(* Schneider Machine Expert - Basic project Prototype 3, file version 2.7.0.0 *)
(* ProjectInformations: Name=Nuevo proyecto *)

HARDWARE
  Cpu 0: TM221M16R/G
  EthernetConfiguration: NetworkName=M221, IpAllocationMode=FixedAddress, IpAddress=0.0.0.0, SubnetMask=0.0.0.0
  SerialLineConfiguration: Baud=Baud19200, Parity=ParityEven, DataBits=DataBits8, StopBits=StopBits1, PhysicalMedium=PhysicalMediumRs485, TransmissionMode=TransmissionModeModbusRtu, SlaveId=1, Addressing=SlaveAddressing
  MastTask: UsePeriodScanMode=false, PeriodScan=100
  FastTask: Period=255
  CpuBehavior: StartingMode=StartAsPreviousState, AutoSaveRamOnEeprom=true, WatchdogPeriod=250

SYMBOLS  (address, symbol, comment, settings)
  %M0       START_BUTTON
  %M1       FINISH_BUTTON
  %M2       STOP_BUTTON
  %M3       EMERGENCY_STOP
  %M4       TYPE_2
  %M5       TYPE_3
  %M6       MACHINE_2
  %M7       MACHINE_3
  %M8       ITEM_1
  %M9       DOOR
  %M10      EXIT_PROCESS_SENSOR
  %M11      ITEM_2
  %M12      RESET_BUTTON
  %M13      ALARM_SIREN
  %M14      GREEN_LIGHT
  %M15      YELLOW_LIGHT
  %M16      RED_LIGHT
  %M17      WARNING_LIGHT
  %M18      GRAB_1
  %M19      PROCESS_INIT
  %M20      AUX_CONVEYOR
  %M21      PROCESS_EXIT
  %M22      GRAB_2
  %M100     INIT_1
  %M200     OK
  %S21      SB_INITGRAFCET  "En el estado 1, este bit provoca una inicialización GRAFCET. Los pasos activos se desactivan y los pasos iniciales se activan"
  %X1       STATE_1
  %X2       STATE_2
  %X3       STATE_3
  %X4       STATE_4
  %X5       STATE_5
  %X6       STATE_6
  %X7       STATE_7
  %X8       STATE_8
  %X9       STATE_9
  %X11      STATE_11
  %X12      STATE_12
  %X13      STATE_13
  %X14      STATE_14
  %X15      STATE_15
  %X17      STATE_17
  %X18      STATE_18
  %X19      STATE_19
  %X20      STATE_20
  %MW0      X_1
  %MW1      Y_1
  %MW2      Z_1
  %MW3      X_2
  %MW4      Y_2
  %MW5      Z_2
  %MW6      SET_X_1
  %MW7      SET_Y_1
  %MW8      SET_Z_1
  %MW9      SET_X_2
  %MW10     SET_Y_2
  %MW11     SET_Z_2
  %MW12     M1
  %MW13     M2
  %MW14     M3
  %KF1      X_Y_ZERO  [Value=0]
  %KF4      X_Y_MED  [Value=5.1]
  %KF7      X_Y_MAX  [Value=10]
  %KF10     Z_MAX  [Value=5.9]
  %KF13     Z_MIN  [Value=2.5]
  %KF16     TOL  [Value=0.1]
  %TM0      SECURITY_TIME  [Preset=5, Base=OneSecond]
  %TM1      FINISH_CONEYOR  [Type=TOF, Preset=3, Base=OneSecond]
  %C0       MACHINE_1_INPUT  [Preset=1000]
  %C1       MACHINE_2_INPUT  [Preset=1000]
  %C2       MACHINE_3_INPUT  [Preset=1000]

GRAFCET Grafcet
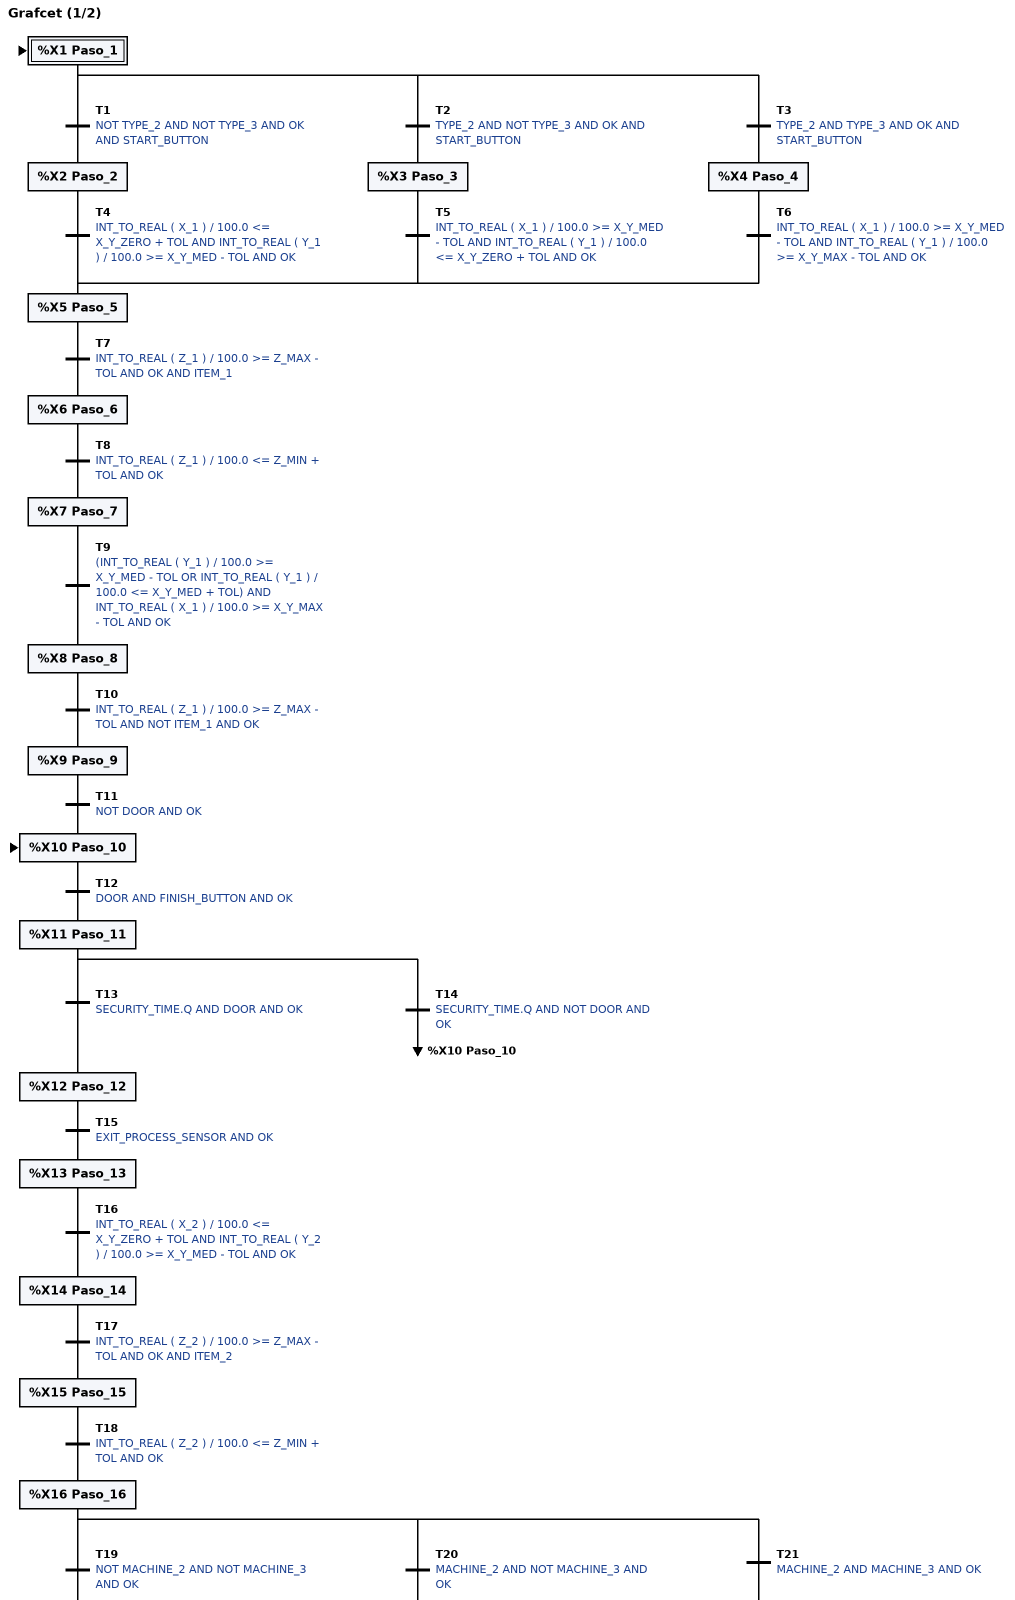
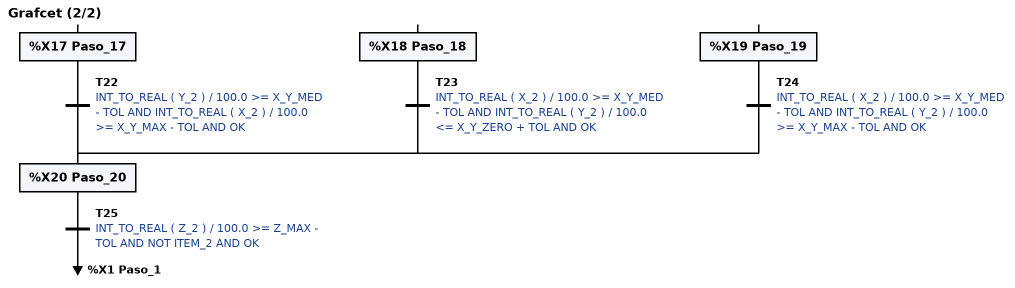
  INITIAL_STEP %X1  (* Paso_1 *)
  STEP %X2  (* Paso_2 *)
  STEP %X3  (* Paso_3 *)
  STEP %X4  (* Paso_4 *)
  STEP %X5  (* Paso_5 *)
  STEP %X6  (* Paso_6 *)
  STEP %X7  (* Paso_7 *)
  STEP %X8  (* Paso_8 *)
  STEP %X9  (* Paso_9 *)
  STEP %X10  (* Paso_10 *)
  STEP %X11  (* Paso_11 *)
  STEP %X12  (* Paso_12 *)
  STEP %X13  (* Paso_13 *)
  STEP %X14  (* Paso_14 *)
  STEP %X15  (* Paso_15 *)
  STEP %X16  (* Paso_16 *)
  STEP %X17  (* Paso_17 *)
  STEP %X18  (* Paso_18 *)
  STEP %X19  (* Paso_19 *)
  STEP %X20  (* Paso_20 *)
  TRANSITION T1 FROM %X1 TO %X2 := NOT TYPE_2 AND NOT TYPE_3 AND OK AND START_BUTTON;
  TRANSITION T2 FROM %X1 TO %X3 := TYPE_2 AND NOT TYPE_3 AND OK AND START_BUTTON;
  TRANSITION T3 FROM %X1 TO %X4 := TYPE_2 AND TYPE_3 AND OK AND START_BUTTON;
  TRANSITION T4 FROM %X2 TO %X5 := INT_TO_REAL ( X_1 ) / 100.0 <= X_Y_ZERO + TOL AND INT_TO_REAL ( Y_1 ) / 100.0 >= X_Y_MED - TOL AND OK;
  TRANSITION T5 FROM %X3 TO %X5 := INT_TO_REAL ( X_1 ) / 100.0 >= X_Y_MED - TOL AND INT_TO_REAL ( Y_1 ) / 100.0 <= X_Y_ZERO + TOL AND OK;
  TRANSITION T6 FROM %X4 TO %X5 := INT_TO_REAL ( X_1 ) / 100.0 >= X_Y_MED - TOL AND INT_TO_REAL ( Y_1 ) / 100.0 >= X_Y_MAX - TOL AND OK;
  TRANSITION T7 FROM %X5 TO %X6 := INT_TO_REAL ( Z_1 ) / 100.0 >= Z_MAX - TOL AND OK AND ITEM_1;
  TRANSITION T8 FROM %X6 TO %X7 := INT_TO_REAL ( Z_1 ) / 100.0 <= Z_MIN + TOL AND OK;
  TRANSITION T9 FROM %X7 TO %X8 := (INT_TO_REAL ( Y_1 ) / 100.0 >= X_Y_MED - TOL OR INT_TO_REAL ( Y_1 ) / 100.0 <= X_Y_MED + TOL) AND INT_TO_REAL ( X_1 ) / 100.0 >= X_Y_MAX - TOL AND OK;
  TRANSITION T10 FROM %X8 TO %X9 := INT_TO_REAL ( Z_1 ) / 100.0 >= Z_MAX - TOL AND NOT ITEM_1 AND OK;
  TRANSITION T11 FROM %X9 TO %X10 := NOT DOOR AND OK;
  TRANSITION T12 FROM %X10 TO %X11 := DOOR AND FINISH_BUTTON AND OK;
  TRANSITION T13 FROM %X11 TO %X12 := SECURITY_TIME.Q AND DOOR AND OK;
  TRANSITION T14 FROM %X11 TO %X10 := SECURITY_TIME.Q AND NOT DOOR AND OK;
  TRANSITION T15 FROM %X12 TO %X13 := EXIT_PROCESS_SENSOR AND OK;
  TRANSITION T16 FROM %X13 TO %X14 := INT_TO_REAL ( X_2 ) / 100.0 <= X_Y_ZERO + TOL AND INT_TO_REAL ( Y_2 ) / 100.0 >= X_Y_MED - TOL AND OK;
  TRANSITION T17 FROM %X14 TO %X15 := INT_TO_REAL ( Z_2 ) / 100.0 >= Z_MAX - TOL AND OK AND ITEM_2;
  TRANSITION T18 FROM %X15 TO %X16 := INT_TO_REAL ( Z_2 ) / 100.0 <= Z_MIN + TOL AND OK;
  TRANSITION T19 FROM %X16 TO %X17 := NOT MACHINE_2 AND NOT MACHINE_3 AND OK;
  TRANSITION T20 FROM %X16 TO %X18 := MACHINE_2 AND NOT MACHINE_3 AND OK;
  TRANSITION T21 FROM %X16 TO %X19 := MACHINE_2 AND MACHINE_3 AND OK;
  TRANSITION T22 FROM %X17 TO %X20 := INT_TO_REAL ( Y_2 ) / 100.0 >= X_Y_MED - TOL AND INT_TO_REAL ( X_2 ) / 100.0 >= X_Y_MAX - TOL AND OK;
  TRANSITION T23 FROM %X18 TO %X20 := INT_TO_REAL ( X_2 ) / 100.0 >= X_Y_MED - TOL AND INT_TO_REAL ( Y_2 ) / 100.0 <= X_Y_ZERO + TOL AND OK;
  TRANSITION T24 FROM %X19 TO %X20 := INT_TO_REAL ( X_2 ) / 100.0 >= X_Y_MED - TOL AND INT_TO_REAL ( Y_2 ) / 100.0 >= X_Y_MAX - TOL AND OK;
  TRANSITION T25 FROM %X20 TO %X1 := INT_TO_REAL ( Z_2 ) / 100.0 >= Z_MAX - TOL AND NOT ITEM_2 AND OK;

TRANSITION T1 (%X1 -> %X2) 
  (* SectionNumber=0 *)

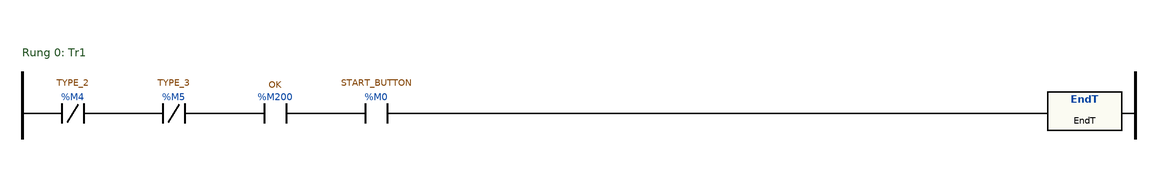

// Rung 0: Tr1
  LDN %M4                 (* TYPE_2 *)
  ANDN %M5                (* TYPE_3 *)
  AND %M200               (* OK *)
  AND %M0                 (* START_BUTTON *)
  ENDT
  // as ST:
  //   TRANSITION := NOT TYPE_2 AND NOT TYPE_3 AND OK AND START_BUTTON;

TRANSITION T2 (%X1 -> %X3) 
  (* SectionNumber=0 *)

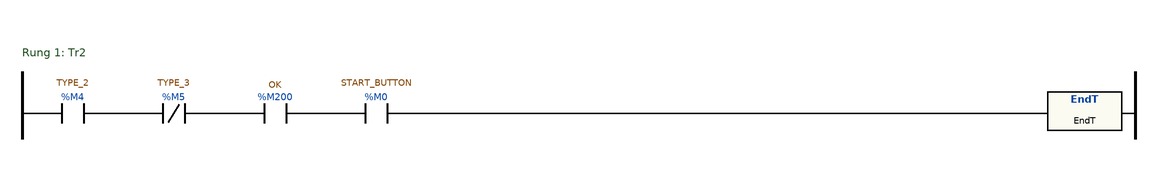

// Rung 1: Tr2
  LD %M4                  (* TYPE_2 *)
  ANDN %M5                (* TYPE_3 *)
  AND %M200               (* OK *)
  AND %M0                 (* START_BUTTON *)
  ENDT
  // as ST:
  //   TRANSITION := TYPE_2 AND NOT TYPE_3 AND OK AND START_BUTTON;

TRANSITION T3 (%X1 -> %X4) 
  (* SectionNumber=0 *)

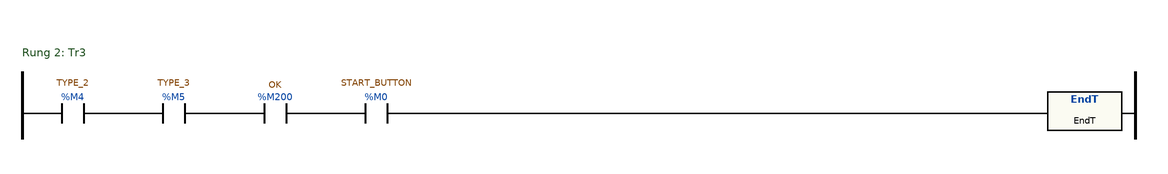

// Rung 2: Tr3
  LD %M4                  (* TYPE_2 *)
  AND %M5                 (* TYPE_3 *)
  AND %M200               (* OK *)
  AND %M0                 (* START_BUTTON *)
  ENDT
  // as ST:
  //   TRANSITION := TYPE_2 AND TYPE_3 AND OK AND START_BUTTON;

TRANSITION T4 (%X2 -> %X5) 
  (* SectionNumber=0 *)

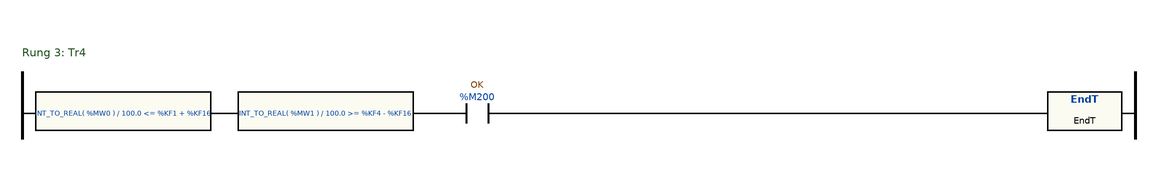

// Rung 3: Tr4
  LD 1
  AND [ INT_TO_REAL ( %MW0 ) / 100.0 <= %KF1 + %KF16 ](* X_1, X_Y_ZERO, TOL *)
  AND [ INT_TO_REAL ( %MW1 ) / 100.0 >= %KF4 - %KF16 ](* Y_1, X_Y_MED, TOL *)
  AND %M200               (* OK *)
  ENDT
  // as ST:
  //   TRANSITION := INT_TO_REAL ( X_1 ) / 100.0 <= X_Y_ZERO + TOL AND INT_TO_REAL ( Y_1 ) / 100.0 >= X_Y_MED - TOL AND OK;

TRANSITION T5 (%X3 -> %X5) 
  (* SectionNumber=0 *)

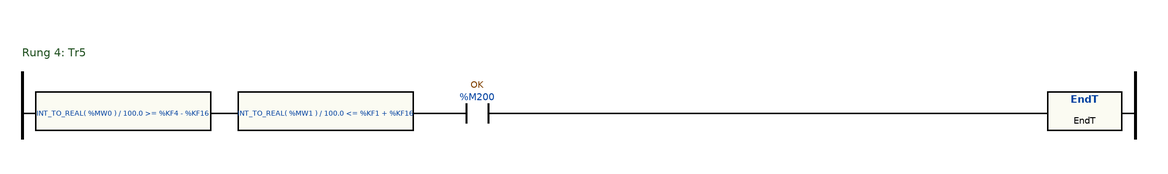

// Rung 4: Tr5
  LD 1
  AND [ INT_TO_REAL ( %MW0 ) / 100.0 >= %KF4 - %KF16 ](* X_1, X_Y_MED, TOL *)
  AND [ INT_TO_REAL ( %MW1 ) / 100.0 <= %KF1 + %KF16 ](* Y_1, X_Y_ZERO, TOL *)
  AND %M200               (* OK *)
  ENDT
  // as ST:
  //   TRANSITION := INT_TO_REAL ( X_1 ) / 100.0 >= X_Y_MED - TOL AND INT_TO_REAL ( Y_1 ) / 100.0 <= X_Y_ZERO + TOL AND OK;

TRANSITION T6 (%X4 -> %X5) 
  (* SectionNumber=0 *)

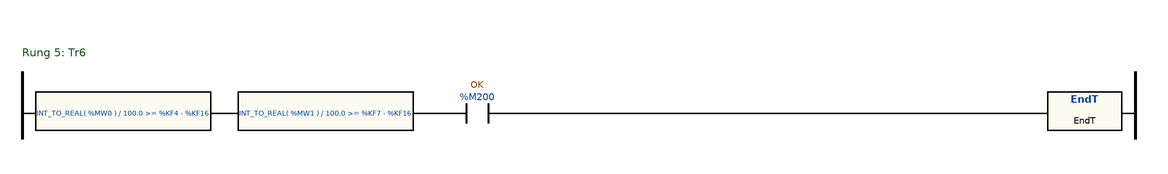

// Rung 5: Tr6
  LD 1
  AND [ INT_TO_REAL ( %MW0 ) / 100.0 >= %KF4 - %KF16 ](* X_1, X_Y_MED, TOL *)
  AND [ INT_TO_REAL ( %MW1 ) / 100.0 >= %KF7 - %KF16 ](* Y_1, X_Y_MAX, TOL *)
  AND %M200               (* OK *)
  ENDT
  // as ST:
  //   TRANSITION := INT_TO_REAL ( X_1 ) / 100.0 >= X_Y_MED - TOL AND INT_TO_REAL ( Y_1 ) / 100.0 >= X_Y_MAX - TOL AND OK;

TRANSITION T7 (%X5 -> %X6) 
  (* SectionNumber=0 *)

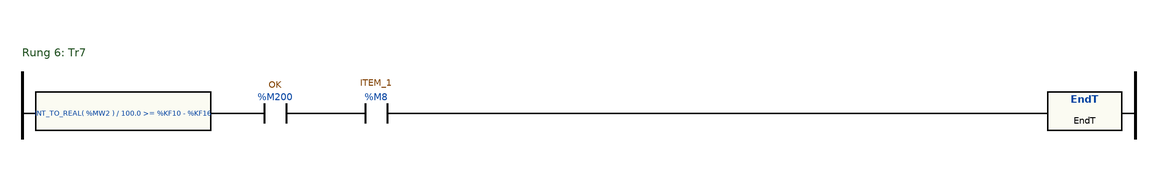

// Rung 6: Tr7
  LD 1
  AND [ INT_TO_REAL ( %MW2 ) / 100.0 >= %KF10 - %KF16 ](* Z_1, Z_MAX, TOL *)
  AND %M200               (* OK *)
  AND %M8                 (* ITEM_1 *)
  ENDT
  // as ST:
  //   TRANSITION := INT_TO_REAL ( Z_1 ) / 100.0 >= Z_MAX - TOL AND OK AND ITEM_1;

TRANSITION T8 (%X6 -> %X7) 
  (* SectionNumber=0 *)

// Rung 7: Tr8
  LD 1
  AND [ INT_TO_REAL ( %MW2 ) / 100.0 <= %KF13 + %KF16 ](* Z_1, Z_MIN, TOL *)
  AND %M200               (* OK *)
  ENDT
  // as ST:
  //   TRANSITION := INT_TO_REAL ( Z_1 ) / 100.0 <= Z_MIN + TOL AND OK;

TRANSITION T9 (%X7 -> %X8) 
  (* SectionNumber=0 *)

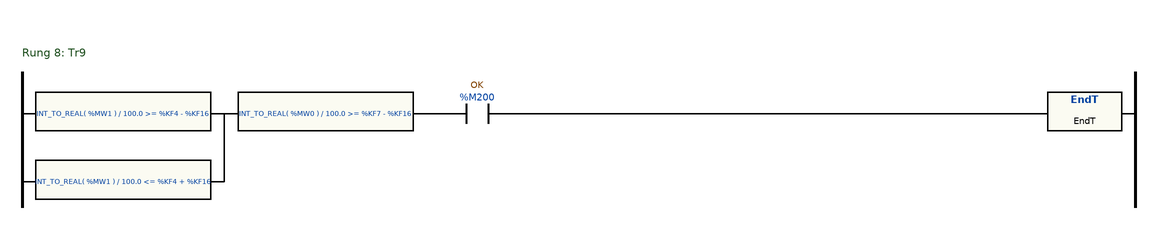

// Rung 8: Tr9
  LD 1
  AND [ INT_TO_REAL ( %MW1 ) / 100.0 >= %KF4 - %KF16 ](* Y_1, X_Y_MED, TOL *)
  OR [ INT_TO_REAL ( %MW1 ) / 100.0 <= %KF4 + %KF16 ](* Y_1, X_Y_MED, TOL *)
  AND [ INT_TO_REAL ( %MW0 ) / 100.0 >= %KF7 - %KF16 ](* X_1, X_Y_MAX, TOL *)
  AND %M200               (* OK *)
  ENDT
  // as ST:
  //   TRANSITION := (INT_TO_REAL ( Y_1 ) / 100.0 >= X_Y_MED - TOL OR INT_TO_REAL ( Y_1 ) / 100.0 <= X_Y_MED + TOL) AND INT_TO_REAL ( X_1 ) / 100.0 >= X_Y_MAX - TOL AND OK;

TRANSITION T10 (%X8 -> %X9) 
  (* SectionNumber=0 *)

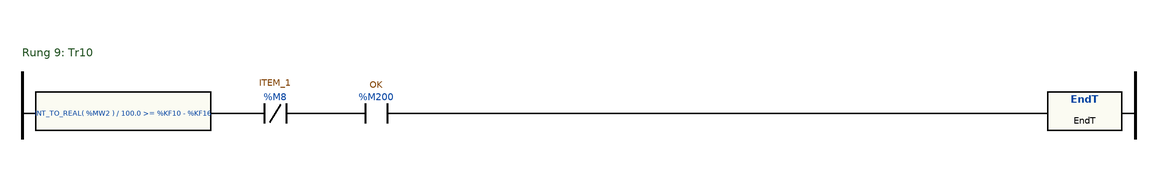

// Rung 9: Tr10
  LD 1
  AND [ INT_TO_REAL ( %MW2 ) / 100.0 >= %KF10 - %KF16 ](* Z_1, Z_MAX, TOL *)
  ANDN %M8                (* ITEM_1 *)
  AND %M200               (* OK *)
  ENDT
  // as ST:
  //   TRANSITION := INT_TO_REAL ( Z_1 ) / 100.0 >= Z_MAX - TOL AND NOT ITEM_1 AND OK;

TRANSITION T11 (%X9 -> %X10) 
  (* SectionNumber=0 *)

// Rung 10: Tr11
  LDN %M9                 (* DOOR *)
  AND %M200               (* OK *)
  ENDT
  // as ST:
  //   TRANSITION := NOT DOOR AND OK;

TRANSITION T12 (%X10 -> %X11) 
  (* SectionNumber=0 *)

// Rung 11: Tr12
  LD %M9                  (* DOOR *)
  AND %M1                 (* FINISH_BUTTON *)
  AND %M200               (* OK *)
  ENDT
  // as ST:
  //   TRANSITION := DOOR AND FINISH_BUTTON AND OK;

TRANSITION T13 (%X11 -> %X12) 
  (* SectionNumber=0 *)

// Rung 12: Tr13
  LD %TM0.Q               (* SECURITY_TIME *)
  AND %M9                 (* DOOR *)
  AND %M200               (* OK *)
  ENDT
  // as ST:
  //   TRANSITION := SECURITY_TIME.Q AND DOOR AND OK;

TRANSITION T14 (%X11 -> %X10) 
  (* SectionNumber=0 *)

// Rung 13: Tr14
  LD %TM0.Q               (* SECURITY_TIME *)
  ANDN %M9                (* DOOR *)
  AND %M200               (* OK *)
  ENDT
  // as ST:
  //   TRANSITION := SECURITY_TIME.Q AND NOT DOOR AND OK;

TRANSITION T15 (%X12 -> %X13) 
  (* SectionNumber=0 *)

// Rung 14: Tr15
  LD %M10                 (* EXIT_PROCESS_SENSOR *)
  AND %M200               (* OK *)
  ENDT
  // as ST:
  //   TRANSITION := EXIT_PROCESS_SENSOR AND OK;

TRANSITION T16 (%X13 -> %X14) 
  (* SectionNumber=0 *)

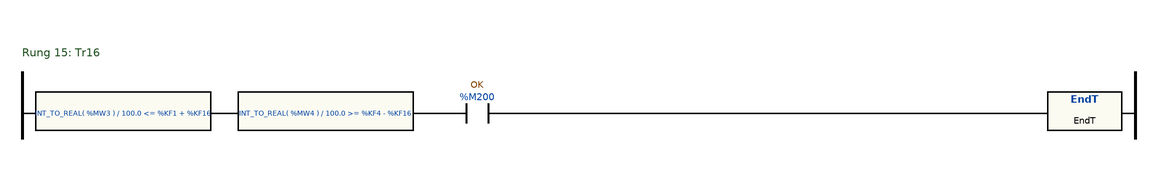

// Rung 15: Tr16
  LD 1
  AND [ INT_TO_REAL ( %MW3 ) / 100.0 <= %KF1 + %KF16 ](* X_2, X_Y_ZERO, TOL *)
  AND [ INT_TO_REAL ( %MW4 ) / 100.0 >= %KF4 - %KF16 ](* Y_2, X_Y_MED, TOL *)
  AND %M200               (* OK *)
  ENDT
  // as ST:
  //   TRANSITION := INT_TO_REAL ( X_2 ) / 100.0 <= X_Y_ZERO + TOL AND INT_TO_REAL ( Y_2 ) / 100.0 >= X_Y_MED - TOL AND OK;

TRANSITION T17 (%X14 -> %X15) 
  (* SectionNumber=0 *)

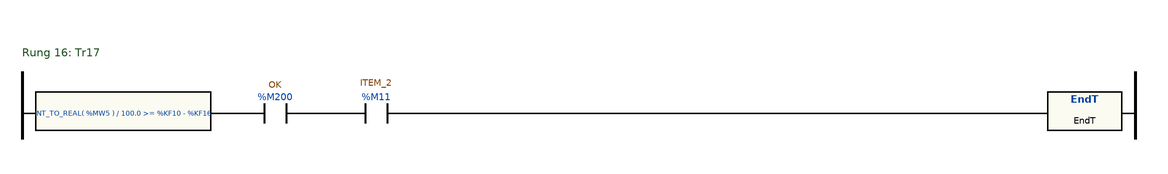

// Rung 16: Tr17
  LD 1
  AND [ INT_TO_REAL ( %MW5 ) / 100.0 >= %KF10 - %KF16 ](* Z_2, Z_MAX, TOL *)
  AND %M200               (* OK *)
  AND %M11                (* ITEM_2 *)
  ENDT
  // as ST:
  //   TRANSITION := INT_TO_REAL ( Z_2 ) / 100.0 >= Z_MAX - TOL AND OK AND ITEM_2;

TRANSITION T18 (%X15 -> %X16) 
  (* SectionNumber=0 *)

// Rung 17: Tr18
  LD 1
  AND [ INT_TO_REAL ( %MW5 ) / 100.0 <= %KF13 + %KF16 ](* Z_2, Z_MIN, TOL *)
  AND %M200               (* OK *)
  ENDT
  // as ST:
  //   TRANSITION := INT_TO_REAL ( Z_2 ) / 100.0 <= Z_MIN + TOL AND OK;

TRANSITION T19 (%X16 -> %X17) 
  (* SectionNumber=0 *)

// Rung 18: Tr19
  LDN %M6                 (* MACHINE_2 *)
  ANDN %M7                (* MACHINE_3 *)
  AND %M200               (* OK *)
  ENDT
  // as ST:
  //   TRANSITION := NOT MACHINE_2 AND NOT MACHINE_3 AND OK;

TRANSITION T20 (%X16 -> %X18) 
  (* SectionNumber=0 *)

// Rung 19: Tr20
  LD %M6                  (* MACHINE_2 *)
  ANDN %M7                (* MACHINE_3 *)
  AND %M200               (* OK *)
  ENDT
  // as ST:
  //   TRANSITION := MACHINE_2 AND NOT MACHINE_3 AND OK;

TRANSITION T21 (%X16 -> %X19) 
  (* SectionNumber=0 *)

// Rung 20: Tr21
  LD %M6                  (* MACHINE_2 *)
  AND %M7                 (* MACHINE_3 *)
  AND %M200               (* OK *)
  ENDT
  // as ST:
  //   TRANSITION := MACHINE_2 AND MACHINE_3 AND OK;

TRANSITION T22 (%X17 -> %X20) 
  (* SectionNumber=0 *)

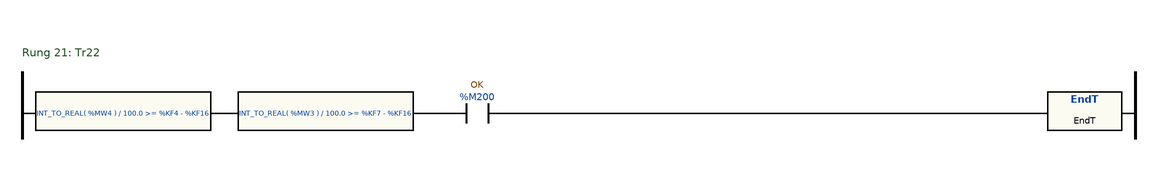

// Rung 21: Tr22
  LD 1
  AND [ INT_TO_REAL ( %MW4 ) / 100.0 >= %KF4 - %KF16 ](* Y_2, X_Y_MED, TOL *)
  AND [ INT_TO_REAL ( %MW3 ) / 100.0 >= %KF7 - %KF16 ](* X_2, X_Y_MAX, TOL *)
  AND %M200               (* OK *)
  ENDT
  // as ST:
  //   TRANSITION := INT_TO_REAL ( Y_2 ) / 100.0 >= X_Y_MED - TOL AND INT_TO_REAL ( X_2 ) / 100.0 >= X_Y_MAX - TOL AND OK;

TRANSITION T23 (%X18 -> %X20) 
  (* SectionNumber=0 *)

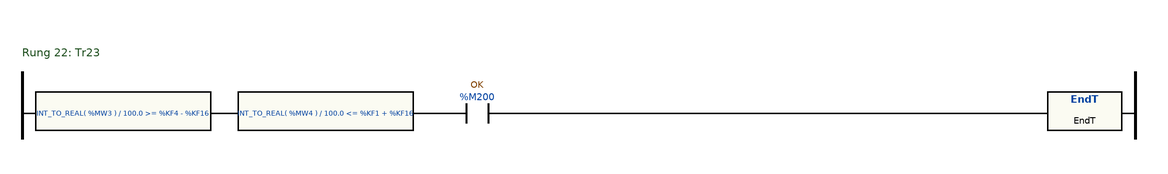

// Rung 22: Tr23
  LD 1
  AND [ INT_TO_REAL ( %MW3 ) / 100.0 >= %KF4 - %KF16 ](* X_2, X_Y_MED, TOL *)
  AND [ INT_TO_REAL ( %MW4 ) / 100.0 <= %KF1 + %KF16 ](* Y_2, X_Y_ZERO, TOL *)
  AND %M200               (* OK *)
  ENDT
  // as ST:
  //   TRANSITION := INT_TO_REAL ( X_2 ) / 100.0 >= X_Y_MED - TOL AND INT_TO_REAL ( Y_2 ) / 100.0 <= X_Y_ZERO + TOL AND OK;

TRANSITION T24 (%X19 -> %X20) 
  (* SectionNumber=0 *)

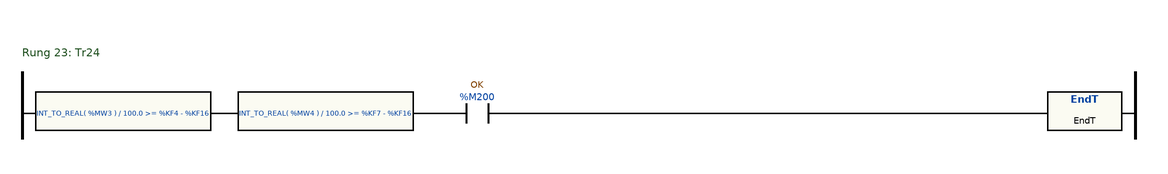

// Rung 23: Tr24
  LD 1
  AND [ INT_TO_REAL ( %MW3 ) / 100.0 >= %KF4 - %KF16 ](* X_2, X_Y_MED, TOL *)
  AND [ INT_TO_REAL ( %MW4 ) / 100.0 >= %KF7 - %KF16 ](* Y_2, X_Y_MAX, TOL *)
  AND %M200               (* OK *)
  ENDT
  // as ST:
  //   TRANSITION := INT_TO_REAL ( X_2 ) / 100.0 >= X_Y_MED - TOL AND INT_TO_REAL ( Y_2 ) / 100.0 >= X_Y_MAX - TOL AND OK;

TRANSITION T25 (%X20 -> %X1) 
  (* SectionNumber=0 *)

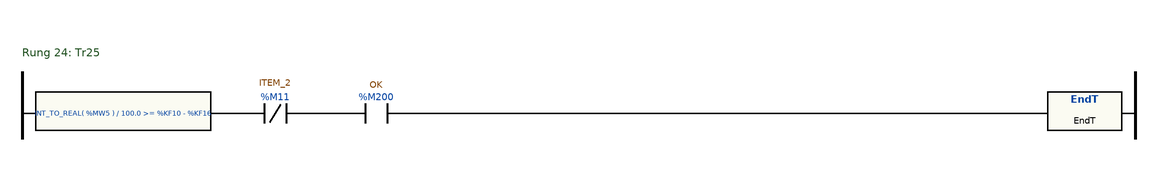

// Rung 24: Tr25
  LD 1
  AND [ INT_TO_REAL ( %MW5 ) / 100.0 >= %KF10 - %KF16 ](* Z_2, Z_MAX, TOL *)
  ANDN %M11               (* ITEM_2 *)
  AND %M200               (* OK *)
  ENDT
  // as ST:
  //   TRANSITION := INT_TO_REAL ( Z_2 ) / 100.0 >= Z_MAX - TOL AND NOT ITEM_2 AND OK;

POU Actions
  (* SectionNumber=22 *)

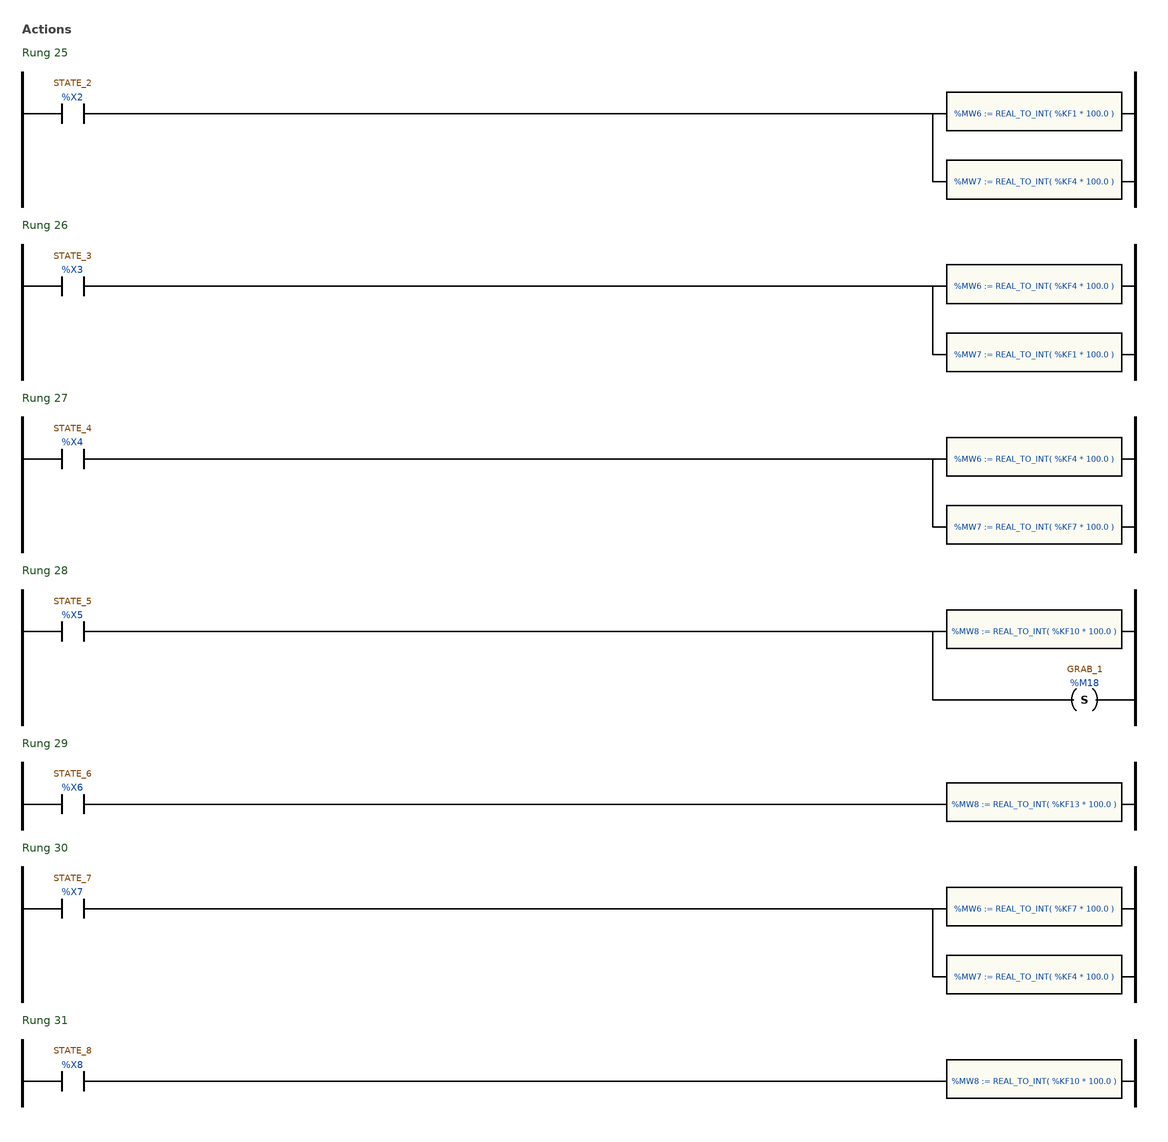

// Rung 25
  LD %X2                  (* STATE_2 *)
  [ %MW6 := REAL_TO_INT ( %KF1 * 100.0 ) ](* SET_X_1, X_Y_ZERO *)
  [ %MW7 := REAL_TO_INT ( %KF4 * 100.0 ) ](* SET_Y_1, X_Y_MED *)
  // as ST:
  //   IF STATE_2 THEN SET_X_1 := REAL_TO_INT ( X_Y_ZERO * 100.0 ); END_IF;
  //   IF STATE_2 THEN SET_Y_1 := REAL_TO_INT ( X_Y_MED * 100.0 ); END_IF;

// Rung 26
  LD %X3                  (* STATE_3 *)
  [ %MW6 := REAL_TO_INT ( %KF4 * 100.0 ) ](* SET_X_1, X_Y_MED *)
  [ %MW7 := REAL_TO_INT ( %KF1 * 100.0 ) ](* SET_Y_1, X_Y_ZERO *)
  // as ST:
  //   IF STATE_3 THEN SET_X_1 := REAL_TO_INT ( X_Y_MED * 100.0 ); END_IF;
  //   IF STATE_3 THEN SET_Y_1 := REAL_TO_INT ( X_Y_ZERO * 100.0 ); END_IF;

// Rung 27
  LD %X4                  (* STATE_4 *)
  [ %MW6 := REAL_TO_INT ( %KF4 * 100.0 ) ](* SET_X_1, X_Y_MED *)
  [ %MW7 := REAL_TO_INT ( %KF7 * 100.0 ) ](* SET_Y_1, X_Y_MAX *)
  // as ST:
  //   IF STATE_4 THEN SET_X_1 := REAL_TO_INT ( X_Y_MED * 100.0 ); END_IF;
  //   IF STATE_4 THEN SET_Y_1 := REAL_TO_INT ( X_Y_MAX * 100.0 ); END_IF;

// Rung 28
  LD %X5                  (* STATE_5 *)
  [ %MW8 := REAL_TO_INT ( %KF10 * 100.0 ) ](* SET_Z_1, Z_MAX *)
  S %M18                  (* GRAB_1 *)
  // as ST:
  //   IF STATE_5 THEN SET_Z_1 := REAL_TO_INT ( Z_MAX * 100.0 ); END_IF;
  //   IF STATE_5 THEN GRAB_1 := TRUE; END_IF;

// Rung 29
  LD %X6                  (* STATE_6 *)
  [ %MW8 := REAL_TO_INT ( %KF13 * 100.0 ) ](* SET_Z_1, Z_MIN *)
  // as ST:
  //   IF STATE_6 THEN SET_Z_1 := REAL_TO_INT ( Z_MIN * 100.0 ); END_IF;

// Rung 30
  LD %X7                  (* STATE_7 *)
  [ %MW6 := REAL_TO_INT ( %KF7 * 100.0 ) ](* SET_X_1, X_Y_MAX *)
  [ %MW7 := REAL_TO_INT ( %KF4 * 100.0 ) ](* SET_Y_1, X_Y_MED *)
  // as ST:
  //   IF STATE_7 THEN SET_X_1 := REAL_TO_INT ( X_Y_MAX * 100.0 ); END_IF;
  //   IF STATE_7 THEN SET_Y_1 := REAL_TO_INT ( X_Y_MED * 100.0 ); END_IF;

// Rung 31
  LD %X8                  (* STATE_8 *)
  [ %MW8 := REAL_TO_INT ( %KF10 * 100.0 ) ](* SET_Z_1, Z_MAX *)
  // as ST:
  //   IF STATE_8 THEN SET_Z_1 := REAL_TO_INT ( Z_MAX * 100.0 ); END_IF;

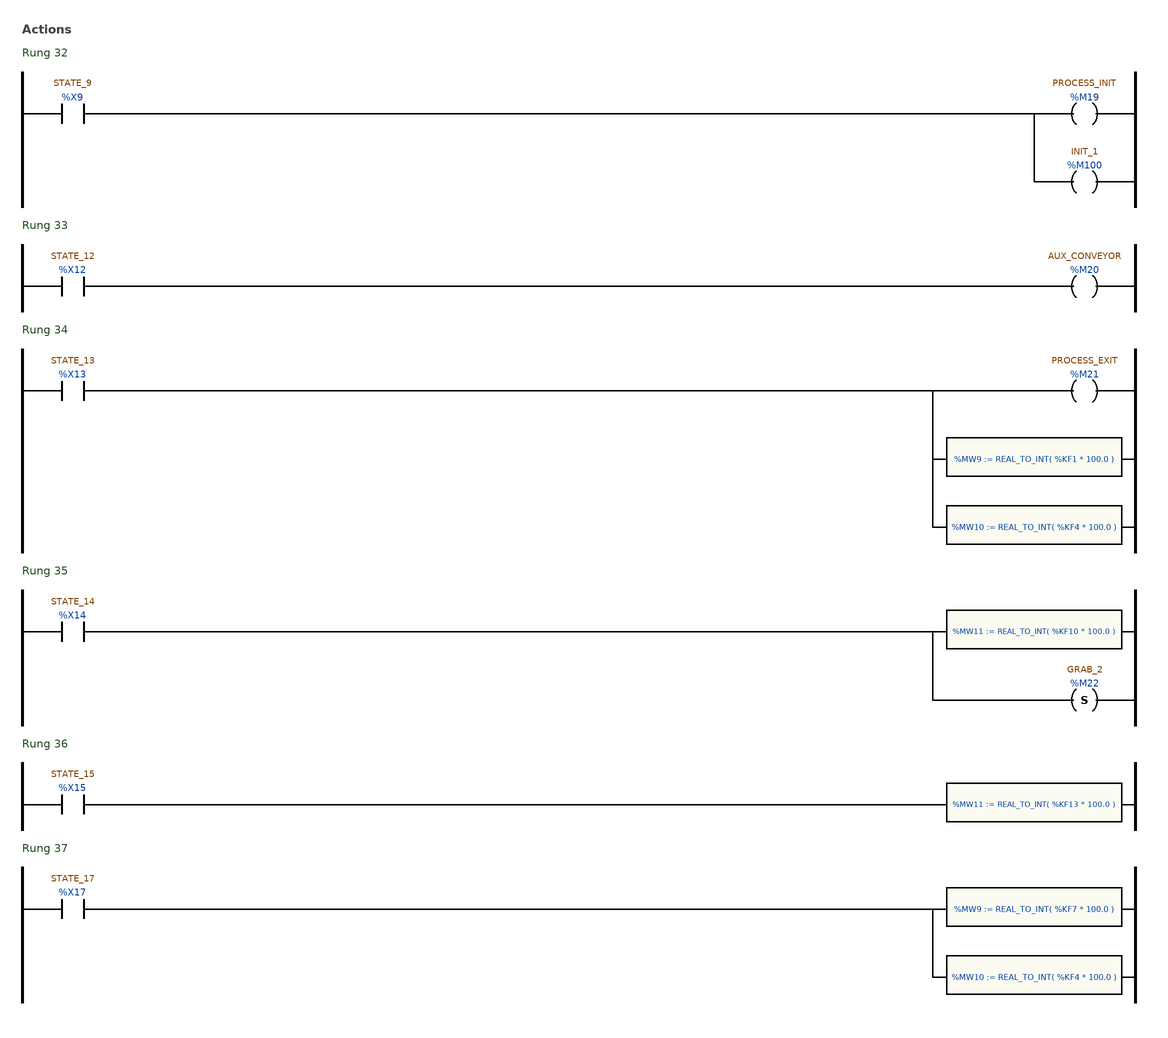

// Rung 32
  LD %X9                  (* STATE_9 *)
  ST %M19                 (* PROCESS_INIT *)
  ST %M100                (* INIT_1 *)
  // as ST:
  //   PROCESS_INIT := STATE_9;
  //   INIT_1 := STATE_9;

// Rung 33
  LD %X12                 (* STATE_12 *)
  ST %M20                 (* AUX_CONVEYOR *)
  // as ST:
  //   AUX_CONVEYOR := STATE_12;

// Rung 34
  LD %X13                 (* STATE_13 *)
  ST %M21                 (* PROCESS_EXIT *)
  [ %MW9 := REAL_TO_INT ( %KF1 * 100.0 ) ](* SET_X_2, X_Y_ZERO *)
  [ %MW10 := REAL_TO_INT ( %KF4 * 100.0 ) ](* SET_Y_2, X_Y_MED *)
  // as ST:
  //   PROCESS_EXIT := STATE_13;
  //   IF STATE_13 THEN SET_X_2 := REAL_TO_INT ( X_Y_ZERO * 100.0 ); END_IF;
  //   IF STATE_13 THEN SET_Y_2 := REAL_TO_INT ( X_Y_MED * 100.0 ); END_IF;

// Rung 35
  LD %X14                 (* STATE_14 *)
  [ %MW11 := REAL_TO_INT ( %KF10 * 100.0 ) ](* SET_Z_2, Z_MAX *)
  S %M22                  (* GRAB_2 *)
  // as ST:
  //   IF STATE_14 THEN SET_Z_2 := REAL_TO_INT ( Z_MAX * 100.0 ); END_IF;
  //   IF STATE_14 THEN GRAB_2 := TRUE; END_IF;

// Rung 36
  LD %X15                 (* STATE_15 *)
  [ %MW11 := REAL_TO_INT ( %KF13 * 100.0 ) ](* SET_Z_2, Z_MIN *)
  // as ST:
  //   IF STATE_15 THEN SET_Z_2 := REAL_TO_INT ( Z_MIN * 100.0 ); END_IF;

// Rung 37
  LD %X17                 (* STATE_17 *)
  [ %MW9 := REAL_TO_INT ( %KF7 * 100.0 ) ](* SET_X_2, X_Y_MAX *)
  [ %MW10 := REAL_TO_INT ( %KF4 * 100.0 ) ](* SET_Y_2, X_Y_MED *)
  // as ST:
  //   IF STATE_17 THEN SET_X_2 := REAL_TO_INT ( X_Y_MAX * 100.0 ); END_IF;
  //   IF STATE_17 THEN SET_Y_2 := REAL_TO_INT ( X_Y_MED * 100.0 ); END_IF;

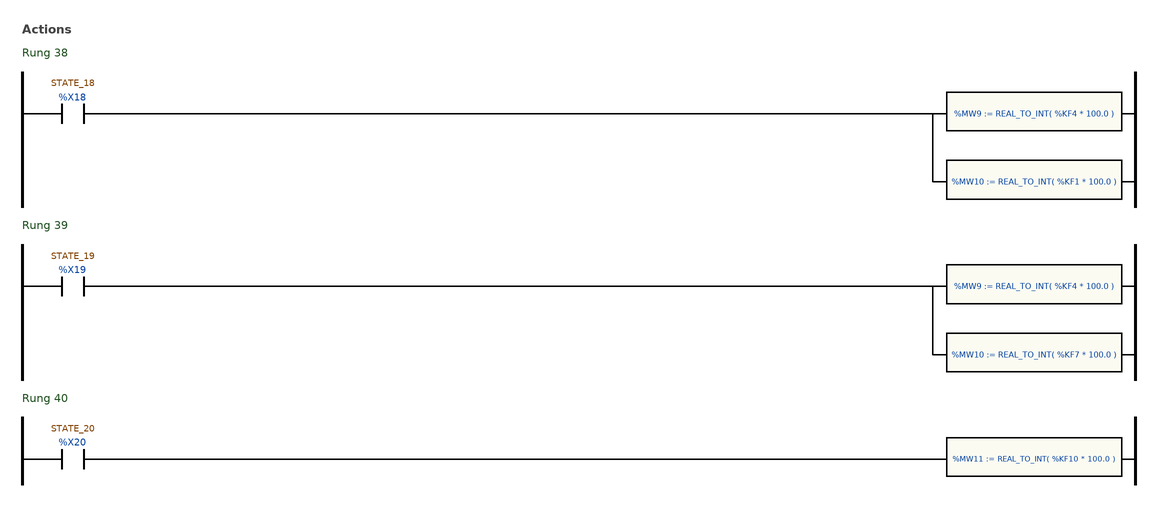

// Rung 38
  LD %X18                 (* STATE_18 *)
  [ %MW9 := REAL_TO_INT ( %KF4 * 100.0 ) ](* SET_X_2, X_Y_MED *)
  [ %MW10 := REAL_TO_INT ( %KF1 * 100.0 ) ](* SET_Y_2, X_Y_ZERO *)
  // as ST:
  //   IF STATE_18 THEN SET_X_2 := REAL_TO_INT ( X_Y_MED * 100.0 ); END_IF;
  //   IF STATE_18 THEN SET_Y_2 := REAL_TO_INT ( X_Y_ZERO * 100.0 ); END_IF;

// Rung 39
  LD %X19                 (* STATE_19 *)
  [ %MW9 := REAL_TO_INT ( %KF4 * 100.0 ) ](* SET_X_2, X_Y_MED *)
  [ %MW10 := REAL_TO_INT ( %KF7 * 100.0 ) ](* SET_Y_2, X_Y_MAX *)
  // as ST:
  //   IF STATE_19 THEN SET_X_2 := REAL_TO_INT ( X_Y_MED * 100.0 ); END_IF;
  //   IF STATE_19 THEN SET_Y_2 := REAL_TO_INT ( X_Y_MAX * 100.0 ); END_IF;

// Rung 40
  LD %X20                 (* STATE_20 *)
  [ %MW11 := REAL_TO_INT ( %KF10 * 100.0 ) ](* SET_Z_2, Z_MAX *)
  // as ST:
  //   IF STATE_20 THEN SET_Z_2 := REAL_TO_INT ( Z_MAX * 100.0 ); END_IF;

POU Init conditions
  (* SectionNumber=23 *)

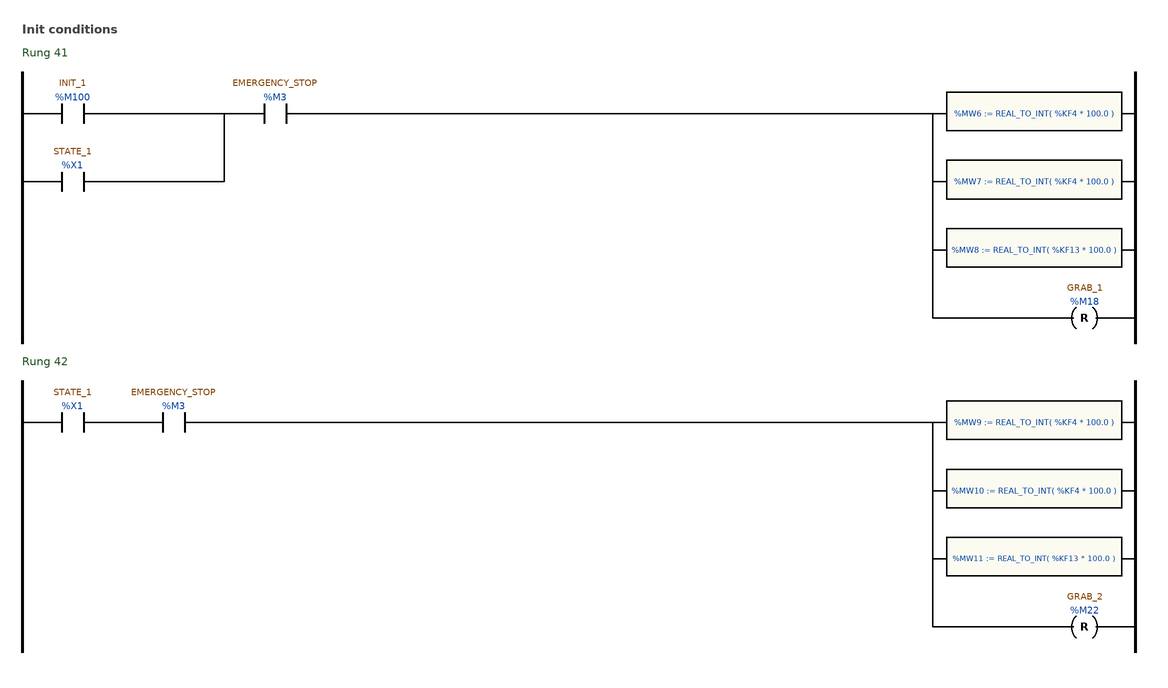

// Rung 41
  LD %M100                (* INIT_1 *)
  OR %X1                  (* STATE_1 *)
  AND %M3                 (* EMERGENCY_STOP *)
  [ %MW6 := REAL_TO_INT ( %KF4 * 100.0 ) ](* SET_X_1, X_Y_MED *)
  [ %MW7 := REAL_TO_INT ( %KF4 * 100.0 ) ](* SET_Y_1, X_Y_MED *)
  [ %MW8 := REAL_TO_INT ( %KF13 * 100.0 ) ](* SET_Z_1, Z_MIN *)
  R %M18                  (* GRAB_1 *)
  // as ST:
  //   IF (INIT_1 OR STATE_1) AND EMERGENCY_STOP THEN SET_X_1 := REAL_TO_INT ( X_Y_MED * 100.0 ); END_IF;
  //   IF (INIT_1 OR STATE_1) AND EMERGENCY_STOP THEN SET_Y_1 := REAL_TO_INT ( X_Y_MED * 100.0 ); END_IF;
  //   IF (INIT_1 OR STATE_1) AND EMERGENCY_STOP THEN SET_Z_1 := REAL_TO_INT ( Z_MIN * 100.0 ); END_IF;
  //   IF (INIT_1 OR STATE_1) AND EMERGENCY_STOP THEN GRAB_1 := FALSE; END_IF;

// Rung 42
  LD %X1                  (* STATE_1 *)
  AND %M3                 (* EMERGENCY_STOP *)
  [ %MW9 := REAL_TO_INT ( %KF4 * 100.0 ) ](* SET_X_2, X_Y_MED *)
  [ %MW10 := REAL_TO_INT ( %KF4 * 100.0 ) ](* SET_Y_2, X_Y_MED *)
  [ %MW11 := REAL_TO_INT ( %KF13 * 100.0 ) ](* SET_Z_2, Z_MIN *)
  R %M22                  (* GRAB_2 *)
  // as ST:
  //   IF STATE_1 AND EMERGENCY_STOP THEN SET_X_2 := REAL_TO_INT ( X_Y_MED * 100.0 ); END_IF;
  //   IF STATE_1 AND EMERGENCY_STOP THEN SET_Y_2 := REAL_TO_INT ( X_Y_MED * 100.0 ); END_IF;
  //   IF STATE_1 AND EMERGENCY_STOP THEN SET_Z_2 := REAL_TO_INT ( Z_MIN * 100.0 ); END_IF;
  //   IF STATE_1 AND EMERGENCY_STOP THEN GRAB_2 := FALSE; END_IF;

POU Timers and counters
  (* SectionNumber=24 *)

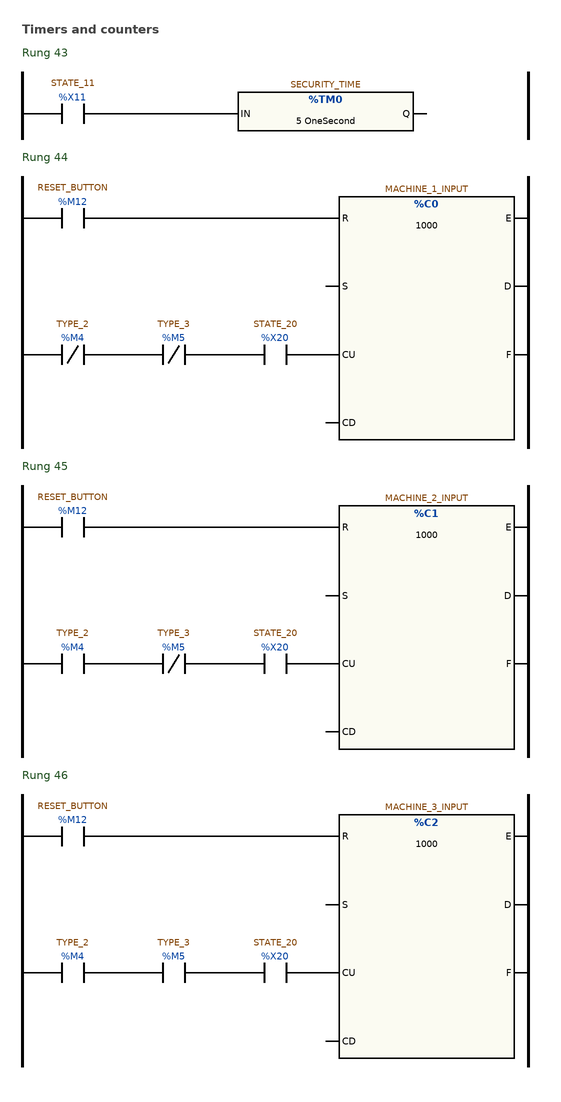

// Rung 43
  BLK %TM0                (* SECURITY_TIME *)
  LD %X11                 (* STATE_11 *)
  IN
  END_BLK
  // as ST:
  //   SECURITY_TIME(IN := STATE_11);

// Rung 44
  BLK %C0                 (* MACHINE_1_INPUT *)
  LD %M12                 (* RESET_BUTTON *)
  R
  LDN %M4                 (* TYPE_2 *)
  ANDN %M5                (* TYPE_3 *)
  AND %X20                (* STATE_20 *)
  CU
  END_BLK
  // as ST:
  //   MACHINE_1_INPUT(R := RESET_BUTTON, CU := NOT TYPE_2 AND NOT TYPE_3 AND STATE_20);

// Rung 45
  BLK %C1                 (* MACHINE_2_INPUT *)
  LD %M12                 (* RESET_BUTTON *)
  R
  LD %M4                  (* TYPE_2 *)
  ANDN %M5                (* TYPE_3 *)
  AND %X20                (* STATE_20 *)
  CU
  END_BLK
  // as ST:
  //   MACHINE_2_INPUT(R := RESET_BUTTON, CU := TYPE_2 AND NOT TYPE_3 AND STATE_20);

// Rung 46
  BLK %C2                 (* MACHINE_3_INPUT *)
  LD %M12                 (* RESET_BUTTON *)
  R
  LD %M4                  (* TYPE_2 *)
  AND %M5                 (* TYPE_3 *)
  AND %X20                (* STATE_20 *)
  CU
  END_BLK
  // as ST:
  //   MACHINE_3_INPUT(R := RESET_BUTTON, CU := TYPE_2 AND TYPE_3 AND STATE_20);

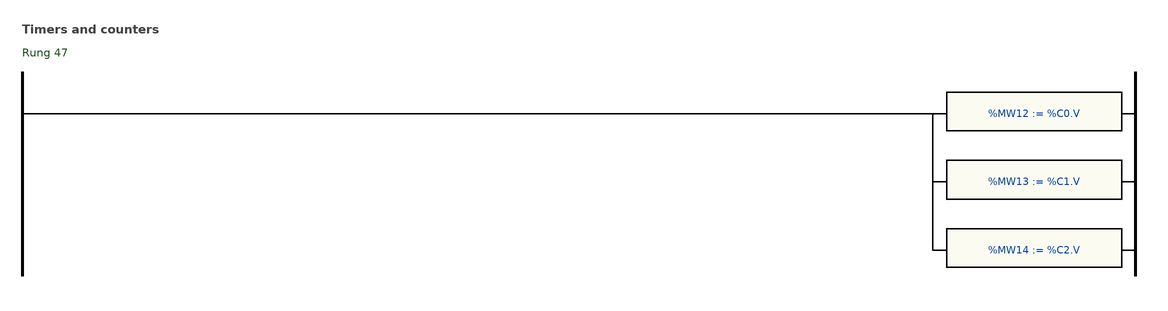

// Rung 47
  LD 1
  [ %MW12 := %C0.V ]      (* M1, MACHINE_1_INPUT *)
  [ %MW13 := %C1.V ]      (* M2, MACHINE_2_INPUT *)
  [ %MW14 := %C2.V ]      (* M3, MACHINE_3_INPUT *)
  // as ST:
  //   M1 := MACHINE_1_INPUT.V;
  //   M2 := MACHINE_2_INPUT.V;
  //   M3 := MACHINE_3_INPUT.V;

POU Buttons
  (* SectionNumber=25 *)

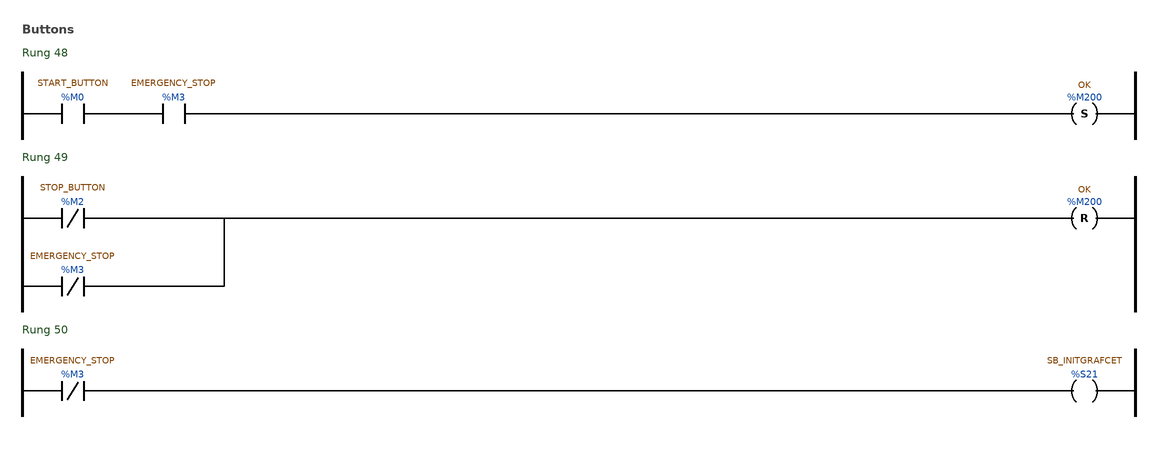

// Rung 48
  LD %M0                  (* START_BUTTON *)
  AND %M3                 (* EMERGENCY_STOP *)
  S %M200                 (* OK *)
  // as ST:
  //   IF START_BUTTON AND EMERGENCY_STOP THEN OK := TRUE; END_IF;

// Rung 49
  LDN %M2                 (* STOP_BUTTON *)
  ORN %M3                 (* EMERGENCY_STOP *)
  R %M200                 (* OK *)
  // as ST:
  //   IF NOT STOP_BUTTON OR NOT EMERGENCY_STOP THEN OK := FALSE; END_IF;

// Rung 50
  LDN %M3                 (* EMERGENCY_STOP *)
  ST %S21                 (* SB_INITGRAFCET *)
  // as ST:
  //   SB_INITGRAFCET := NOT EMERGENCY_STOP;

POU Lights & Warnings
  (* SectionNumber=26 *)

